{attribute 'linkalways'} 
{attribute 'no_explicit_call' := 'This FB is a CLASS and must be accessed using methods or properties'}
{attribute 'enable_dynamic_creation'}
FUNCTION_BLOCK _ETcVnNbc EXTENDS EnumDatatypeBase
VAR
	localData : ETcVnNbc;
	activeData : REFERENCE TO ETcVnNbc;
	enumBaseDatatype : _UDINT(localData);
END_VAR

METHOD PRIVATE AddLocalEnumeration
VAR_INPUT
	Enumeration : T_MAXSTRING;
	Value : ETcVnNbc;
END_VAR
AddEnumeration(Enumeration, Value);
END_METHOD

PROPERTY PUBLIC Address : PVOID
GET
Address := ADR(activeData);
END_GET
END_PROPERTY

METHOD PUBLIC ClearReference
VAR_INPUT
END_VAR
activeData REF= localData;
SetBaseDatatypeReference();
END_METHOD

METHOD PUBLIC Clone : I_Datatype
VAR
    pClone : POINTER TO _ETcVnNbc;
END_VAR
pClone := __NEW(_ETcVnNbc(InitialValue := Value));
Clone := pClone^;
END_METHOD

METHOD FB_init : BOOL
VAR_INPUT
	bInitRetains : BOOL; // if TRUE, the retain variables are initialized (warm start / cold start)
	bInCopyCode : BOOL;  // if TRUE, the instance afterwards gets moved into the copy code (online change)
	InitialValue : ETcVnNbc;
END_VAR
localData := InitialValue;
AddBaseDatatype(enumBaseDatatype);
ClearReference();

AddLocalEnumeration('TCVN_NBC_CLASSIFIER', ETcVnNbc.TCVN_NBC_CLASSIFIER);
AddLocalEnumeration('TCVN_NBC_NOVELTY_DETECTOR', ETcVnNbc.TCVN_NBC_NOVELTY_DETECTOR);
END_METHOD

PROPERTY PUBLIC Identifier : T_MAXSTRING
GET
Identifier := 'ETcVnNbc';
END_GET
END_PROPERTY

METHOD IsEnumeratorValueEqual : BOOL
VAR_INPUT
	Enumerator : I_KeyValueForwardEnumerator;
END_VAR
VAR
	storedValue : ETcVnNbc;
END_VAR
IF NOT Enumerator.TryGet(storedValue) THEN
	RETURN;
END_IF

IsEnumeratorValueEqual := storedValue = activeData;
END_METHOD

METHOD PUBLIC MakeReferenceTo
VAR_INPUT
	ReferenceTarget : REFERENCE TO ETcVnNbc;
END_VAR
activeData REF= ReferenceTarget;
SetBaseDatatypeReference();
END_METHOD

METHOD PROTECTED SetBaseDatatypeReference
VAR_INPUT
END_VAR
enumBaseDatatype.MakeReferenceTo(activeData);
END_METHOD

PROPERTY PUBLIC Size : UDINT
GET
Size := SIZEOF(activeData);
END_GET
END_PROPERTY

METHOD TryMakeReferenceTo : BOOL
VAR_INPUT
	Target : I_Datatype;
END_VAR
VAR
	targetAsEnum : I_EnumDatatype;
	pTargetData : POINTER TO ETcVnNbc;
END_VAR
IF NOT Target.TryResolveAsEnumDatatype(targetAsEnum) THEN
	RETURN;
END_IF

IF targetAsEnum.Identifier <> Identifier THEN
	RETURN;
END_IF

pTargetData := Target.Address;
activeData REF= pTargetData^;
SetBaseDatatypeReference();
TryMakeReferenceTo := TRUE;
END_METHOD

PROPERTY PUBLIC Value : ETcVnNbc
GET
Value := activeData;
END_GET
SET
activeData := Value;
END_SET
END_PROPERTY

END_FUNCTION_BLOCK

(* stored: Version 1.1.0.1, ProductVersion 3.1.4024.12
   POU _ETcVnNbc: Id {3c4ecedc-ffab-0c5a-37fe-33dc50e95fe3}, SpecialFunc None
   Folder Constructor: Id {9126b519-868a-073f-228c-f24a21d47e23}
   Folder Private: Id {aa84247b-2521-0411-3cff-0c74634d696f}
   Folder Protected: Id {4fd3b047-5877-032d-1053-1426449ac904}
   Method AddLocalEnumeration: Id {678128e1-72fe-0c8a-2a91-c55347d4c561}
   Property Address: Id {2bd74b5a-2746-0127-0670-1ed8ff487b1f}
   Get Get: Id {62f94aa8-2c22-0abf-38aa-8ad8b46e461b}
   Method ClearReference: Id {9a0df9e4-a661-0bff-1c62-6356515aeb15}
   Method Clone: Id {7b87e092-37c7-0391-129a-c7ad51b6a317}
   Method FB_init: Id {7818b4f0-34a3-0f75-0f17-22099a2a8062}
   Property Identifier: Id {37907f33-f708-023b-1e46-8e4b37454c04}
   Get Get: Id {419bdfca-9d62-0322-1bc2-a5a5e9a3fcb3}
   Method IsEnumeratorValueEqual: Id {09ceb3f4-e357-0d84-385c-62d38860bd8e}
   Method MakeReferenceTo: Id {9a5f3503-da7c-029f-0808-3b9d7a44863e}
   Method SetBaseDatatypeReference: Id {aac468f9-b243-06ac-2808-a7494278f98b}
   Property Size: Id {122b3e7a-a8e5-0322-36e5-02d0554c7874}
   Get Get: Id {40e905a0-0f38-0dc9-2458-d0fd23da6693}
   Method TryMakeReferenceTo: Id {64fec48a-be99-01de-07c4-bbe607e5c578}
   Property Value: Id {8b82242c-239c-0f89-3eba-ad3e05692aef}
   Get Get: Id {22fd280c-a6b9-07f3-3de9-dd9bcaa13e25}
   Set Set: Id {00785422-fdea-03af-157d-ebb94bc1b2f1} *)
